# EPICS substitutions: iocBoot/ioc13bmd_pg1/TomoCollect.substitutions
file "$(CARS)/db/TomoCollect.template"
{
pattern
{    P,       R,     CAMERA,        MCS,       ROTATION,  SAMPLE_X,  SAMPLE_Y,      BEAM_READY,            CLOSE_SHUTTER,        CLOSE_VALUE,        OPEN_SHUTTER,         OPEN_VALUE}
{13BMDPG1:,  TC:,   13BMDPG1:,  13BMD:SIS1:,  13BMD:m38, 13BMD:m85, 13BMD:m90, 13BMA:mono_pid1Locked, 13BMA:CloseBMDShutter.PROC,    1,        13BMA:OpenBMDShutter.PROC,      1}
}
